// TIA Portal project "BTL" (V15)

(* hardware
DEVICE "PC-System_1"  SIMATIC PC station
   slot 0: "SIMATIC PC station"  Rail  SIMATIC PC-Station  V1.0
      slot 125: "Stationmanager"  Station_Manager  V6.0.4
   slot 1: "HMI_RT_1"  WinCC RT Professional  6AV2 105-0xxxx-xxxx  15.0.0.0
DEVICE "S7300/ET200M station_1"  S7-300 station
   slot 0: "Rail_0"  Rail  6ES7 390-1***0-0AA0
   slot 2: "PLC_1"  CPU 314C-2 PN/DP  6ES7 314-6EH04-0AB0  V3.3
      slot 2: "PROFINET interface_1"  PN-IO
         slot 1: "Port_1"  Port
         slot 2: "Port_2"  Port
      slot 5: "DI 24/DO 16_1"  DI24/DO16
      slot 6: "AI 5/AO 2_1"  AI5/AO2
      slot 7: "Count_1"  Counter
      slot 8: "Positioning_1"  Positioning
*)

// ===== PLC "PLC_1"  CPU 314C-2 PN/DP =====

ORGANIZATION_BLOCK "Main"   // OB1, LAD
TITLE = "Main Program Sweep (Cycle)"
{ S7_Optimized_Access := 'FALSE' }
VERSION : 0.1
   VAR_TEMP
      OB1_EV_CLASS : Byte;   // Bits 0-3 = 1 (Coming event), Bits 4-7 = 1 (Event class 1)
      OB1_SCAN_1 : Byte;   // 1 (Cold restart scan 1 of OB 1), 3 (Scan 2-n of OB 1)
      OB1_PRIORITY : Byte;   // Priority of OB Execution
      OB1_OB_NUMBR : Byte;   // 1 (Organization block 1, OB1)
      OB1_RESERVED_1 : Byte;   // Reserved for system
      OB1_RESERVED_2 : Byte;   // Reserved for system
      OB1_PREV_CYCLE : Int;   // Cycle time of previous OB1 scan (milliseconds)
      OB1_MIN_CYCLE : Int;   // Minimum cycle time of OB1 (milliseconds)
      OB1_MAX_CYCLE : Int;   // Maximum cycle time of OB1 (milliseconds)
      OB1_DATE_TIME : Date_And_Time;   // Date and time OB1 started
   END_VAR
BEGIN
END_ORGANIZATION_BLOCK

(* ===== HMI "HMI_RT_1" =====

screen "Screen_1" 1024x768
   SymbolLibrary "Symbol library_1" at 745,86 size 128x191
   SymbolLibrary "Symbol library_2" at 133,633 size 106x75
   SymbolLibrary "Symbol library_3" at 546,637 size 104x71
   SymbolLibrary "Symbol library_4" at 118,479 size 64x58
   SymbolLibrary "Symbol library_5" at 766,589 size 120x120
   SymbolLibrary "Symbol library_6" at 153,351 size 46x70
   SymbolLibrary "Symbol library_7" at 870,589 size 120x120
   SymbolLibrary "Symbol library_8" at 584,478 size 65x59
   SymbolLibrary "Symbol library_9" at 77,102 size 76x45
   TextField "Text field_1" at 85,150 size 63x21; Text 'OPENED'
   TextField "Text field_2" at 87,177 size 61x21; Text 'CLOSED'
   IOField "I/O field_1" at 269,7 size 39x27; FormatPattern 99999999
   IOField "I/O field_2" at 308,7 size 39x27; FormatPattern 99999999
   IOField "I/O field_3" at 347,7 size 39x27; FormatPattern 99999999
   IOField "I/O field_4" at 518,14 size 39x27; FormatPattern 99999999
   IOField "I/O field_5" at 518,48 size 39x27; FormatPattern 99999999
   IOField "I/O field_6" at 518,82 size 39x27; FormatPattern 99999999
   IOField "I/O field_7" at 585,15 size 39x27; FormatPattern 99999999
   IOField "I/O field_8" at 585,49 size 39x27; FormatPattern 99999999
   IOField "I/O field_9" at 585,83 size 39x27; FormatPattern 99999999
   IOField "I/O field_10" at 269,39 size 39x27; FormatPattern 99999999
   IOField "I/O field_11" at 308,39 size 39x27; FormatPattern 99999999
   IOField "I/O field_12" at 347,39 size 39x27; FormatPattern 99999999
   SymbolLibrary "Symbol library_10" at 191,491 size 70x46
   SymbolLibrary "Symbol library_11" at 250,491 size 70x46
   SymbolLibrary "Symbol library_12" at 309,491 size 70x46
   SymbolLibrary "Symbol library_13" at 368,491 size 70x46
   SymbolLibrary "Symbol library_14" at 427,491 size 70x46
   SymbolLibrary "Symbol library_15" at 486,491 size 70x46
   IOField "I/O field_13" at 221,458 size 40x23; FormatPattern 99999999
   IOField "I/O field_14" at 478,457 size 40x23; FormatPattern 99999999
   IOField "I/O field_15" at 483,277 size 40x23; FormatPattern 99999999
   EllipseSegment "Ellipse segment_1" at 188,303 size 60x28
   SymbolLibrary "Symbol library_16" at 641,124 size 53x62
   SymbolLibrary "Symbol library_17" at 573,351 size 42x71
   SymbolLibrary "Symbol library_18" at 200,537 size 30x25
   SymbolLibrary "Symbol library_19" at 72,548 size 131x14
   SymbolLibrary "Symbol library_20" at 547,537 size 30x25
   SymbolLibrary "Symbol library_21" at 572,548 size 131x14
   SymbolLibrary "Symbol library_22" at 701,518 size 73x51
   SymbolLibrary "Symbol library_23" at 0,518 size 73x51
   IOField "I/O field_16" at 695,50 size 39x27; FormatPattern 99999999
   SymbolLibrary "Symbol library_24" at 842,35 size 49x42
   TextField "Text field_3" at 901,98 size 35x21; Text 'High'
   TextField "Text field_4" at 901,194 size 31x21; Text 'Low'
   TextField "Text field_5" at 10,580 size 105x21; Text 'Quat hut am 1'
   TextField "Text field_6" at 673,574 size 105x21; Text 'Quat hut am 2'
   TextField "Text field_8" at 774,719 size 223x21; Text 'Trung tam dieu khien he thong'
   TextField "Text field_7" at 664,27 size 117x21; Text 'Tuoi trong vong'
   TextField "Text field_9" at 629,14 size 26x21; Text '[M]'
   TextField "Text field_10" at 630,48 size 26x21; Text '[M]'
   TextField "Text field_11" at 630,82 size 26x21; Text '[M]'
   TextField "Text field_12" at 557,14 size 25x21; Text '[H]'
   TextField "Text field_13" at 559,49 size 25x21; Text '[H]'
   TextField "Text field_14" at 559,82 size 25x21; Text '[H]'
   TextField "Text field_15" at 403,18 size 108x21; Text 'Dat time tuoi 1'
   TextField "Text field_16" at 403,48 size 108x21; Text 'Dat time tuoi 2'
   TextField "Text field_17" at 403,78 size 108x21; Text 'Dat time tuoi 3'
   TextField "Text field_18" at 168,10 size 95x21; Text 'Ngay hien tai'
   TextField "Text field_19" at 168,38 size 95x21; Text 'Time hien tai'
   TextField "Text field_20" at 73,77 size 74x21; Text 'Motor mai'
   TextField "Text field_21" at 206,434 size 73x21; Text 'CB Do am'
   TextField "Text field_22" at 483,430 size 63x21; Text 'CB Nhiet'
   TextField "Text field_23" at 261,455 size 30x21; Text '[%]'
   TextField "Text field_24" at 518,460 size 34x21; Text '[Do]'
   TextField "Text field_25" at 478,252 size 90x21; Text 'CB anh sang'
   TextField "Text field_26" at 489,304 size 42x21; Text '[LUX]'
   TextField "Text field_27" at 221,277 size 110x21; Text 'Den chieu sang'
   TextField "Text field_28" at 0,261 size 177x21; Text 'Hop dien den chieu sang'
   TextField "Text field_29" at 734,49 size 26x21; Text '[M]'
   TextField "Text field_30" at 103,428 size 79x21; Text 'Gia nhiet 1'
   TextField "Text field_31" at 585,428 size 79x21; Text 'Gia nhiet 2'
   Button "Button_2" at 711,358 size 52x20; TextOff 'Auto'
   Button "Button_3" at 760,358 size 52x20; TextOff 'Manu'
   Button "Button_4" at 711,389 size 52x20; TextOff 'Start'
   Button "Button_5" at 760,389 size 52x20; TextOff 'Stop'
   Button "Button_6" at 710,416 size 104x22; TextOff 'Simulation'
   IOField "I/O field_17" at 890,379 size 41x23; FormatPattern 99999999
   IOField "I/O field_18" at 931,378 size 41x23; FormatPattern 99999999
   IOField "I/O field_19" at 890,425 size 41x23; FormatPattern 99999999
   IOField "I/O field_20" at 931,424 size 41x23; FormatPattern 99999999
   IOField "I/O field_21" at 890,471 size 41x23; FormatPattern 99999999
   IOField "I/O field_22" at 931,470 size 41x23; FormatPattern 99999999
   TextField "Text field_32" at 697,304 size 115x21; Text 'Bang dieu khien'
   TextField "Text field_33" at 878,306 size 118x21; Text 'Cai dat thong so'
   TextField "Text field_34" at 896,331 size 72x21; Text 'cho phep'
   TextField "Text field_35" at 891,357 size 30x21; Text 'Max'
   TextField "Text field_36" at 929,357 size 27x21; Text 'Min'
   TextField "Text field_37" at 893,400 size 30x21; Text 'Max'
   TextField "Text field_38" at 931,400 size 27x21; Text 'Min'
   TextField "Text field_39" at 894,451 size 30x21; Text 'Max'
   TextField "Text field_40" at 932,451 size 27x21; Text 'Min'
   TextField "Text field_41" at 970,381 size 34x21; Text '[Do]'
   TextField "Text field_42" at 974,422 size 39x21; Text '[Lux]'
   TextField "Text field_43" at 977,470 size 30x21; Text '[%]'
   TextField "Text field_44" at 858,378 size 24x21; Text 'ND'
   TextField "Text field_45" at 860,421 size 22x21; Text 'AS'
   TextField "Text field_46" at 860,472 size 24x21; Text 'DA'
   Button "Button_1" at 6,726 size 80x30; TextOff 'Exit'
   SymbolLibrary "Symbol library_25" at 330,637 size 108x76
   TextField "Text field_47" at 143,719 size 48x21; Text 'Xe xuc'
   TextField "Text field_48" at 363,721 size 71x21; Text 'Xe van tai'
   TextField "Text field_49" at 576,717 size 37x21; Text 'Xe ui'
*)